(* IEC 61131-3 sources: com.logicals.lc3.webinar/usRTS_RPMControl_iSOC/src_FB_LIB_SAFE/Convert/WORD, 4 files *)

(* ---- wTRUNC_WORD_TO_BYTE.iecst ---- *)
NAMESPACE logicals.web.standard
NAMESPACE convert

/*
 * Function block wrapper for IEC 61131-3 TO_BYTE<br>
 * IN =  input value (WORD)<br>
 * OUT = IN (BYTE)<br>
 */
FUNCTION_BLOCK wTRUNC_WORD_TO_BYTE
	{ vNameAlignment:="center"; altName:="TRUNC_WORD_TO_BYTE"; bgColor:="DodgerBlue"; width:=180; hideIONames; }
	VAR_INPUT
		IN : WORD;
	END_VAR
	VAR_OUTPUT
		OUT: BYTE;
	END_VAR

	OUT := TO_BYTE(IN:=IN, ENO=>ENO);
END_FUNCTION_BLOCK

END_NAMESPACE
END_NAMESPACE

(* ---- wWORD_TO_DWORD.iecst ---- *)
NAMESPACE logicals.web.standard
NAMESPACE convert

/*
 * Function block wrapper for IEC 61131-3 TO_DWORD<br>
 * IN =  input value (WORD)<br>
 * OUT = IN (DWORD)<br>
 */
FUNCTION_BLOCK wWORD_TO_DWORD
	{ vNameAlignment:="center"; altName:="WORD_TO_DWORD"; bgColor:="DodgerBlue"; width:=140; hideIONames; }
	VAR_INPUT
		IN : WORD;
	END_VAR
	VAR_OUTPUT
		OUT: DWORD;
	END_VAR

	OUT := TO_DWORD(IN:=IN, ENO=>ENO);
END_FUNCTION_BLOCK

END_NAMESPACE
END_NAMESPACE

(* ---- wWORD_TO_LWORD.iecst ---- *)
NAMESPACE logicals.web.standard
NAMESPACE convert

/*
 * Function block wrapper for IEC 61131-3 TO_LWORD<br>
 * IN =  input value (WORD)<br>
 * OUT = IN (LWORD)<br>
 */
FUNCTION_BLOCK wWORD_TO_LWORD
	{ vNameAlignment:="center"; altName:="WORD_TO_LWORD"; bgColor:="DodgerBlue"; width:=140; hideIONames; }
	VAR_INPUT
		IN : WORD;
	END_VAR
	VAR_OUTPUT
		OUT: LWORD;
	END_VAR

	OUT := TO_LWORD(IN:=IN, ENO=>ENO);
END_FUNCTION_BLOCK

END_NAMESPACE
END_NAMESPACE

(* ---- wWORD_TO_UINT.iecst ---- *)
NAMESPACE logicals.web.standard
NAMESPACE convert

/*
 * Function block wrapper for IEC 61131-3 TO_UINT<br>
 * IN =  input value (WORD)<br>
 * OUT = IN (UINT)<br>
 */
FUNCTION_BLOCK wWORD_TO_UINT
	{ vNameAlignment:="center"; altName:="WORD_TO_UINT"; bgColor:="Plum"; width:=140; hideIONames; }
	VAR_INPUT
		IN : WORD;
	END_VAR
	VAR_OUTPUT
		OUT: UINT;
	END_VAR

	OUT := TO_UINT(IN:=IN, ENO=>ENO);
END_FUNCTION_BLOCK

END_NAMESPACE
END_NAMESPACE
